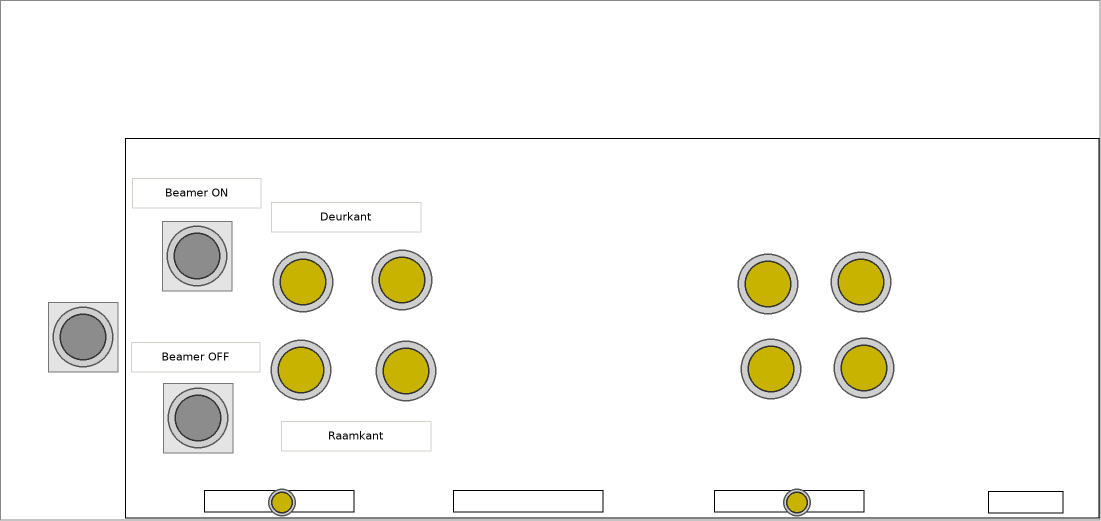
VISUALIZATION Visualization  // 1101x521
    Rectangle (125,138 974x380)
    Lamp1 (268,247 70x70), variable: Lichtsturing.relaisstandDEUR, style: Lamp-Lamp1-Yellow
    Lamp1 (367,245 70x70), variable: Lichtsturing.relaisstandDEUR, style: Lamp-Lamp1-Yellow
    Lamp1 (733,249 70x70), variable: Lichtsturing.relaisstandDEUR, style: Lamp-Lamp1-Yellow
    Lamp1 (826,247 70x70), variable: Lichtsturing.relaisstandDEUR, style: Lamp-Lamp1-Yellow
    Lamp1 (266,335 70x70), variable: Lichtsturing.relaisstandRAAM, style: Lamp-Lamp1-Yellow
    Lamp1 (371,336 70x70), variable: Lichtsturing.relaisstandRAAM, style: Lamp-Lamp1-Yellow
    Lamp1 (736,334 70x70), variable: Lichtsturing.relaisstandRAAM, style: Lamp-Lamp1-Yellow
    Lamp1 (829,333 70x70), variable: Lichtsturing.relaisstandRAAM, style: Lamp-Lamp1-Yellow
    Rectangle (204,490 150x22)
    Rectangle (453,490 150x22)
    Rectangle (714,490 150x22)
    Rectangle (988,491 75x22)
    Lamp1 (266,486 32x33), variable: EnOcean.raam2open, style: Lamp-Lamp1-Yellow
    Lamp1 (781,486 32x33), variable: EnOcean.raam1open, style: Lamp-Lamp1-Yellow
    Textfield (271,202 150x30), "Deurkant"
    Textfield (281,421 150x30), "Raamkant"
    PushSwitch (162,221 70x70), variable: BeamerAANKNOP, behaviour: TOGGLE, style: Switch-PushSwitch-Gray
    Textfield (132,178 129x30), "Beamer ON"
    PushSwitch (163,383 70x70), variable: BeamerUITKNOP, behaviour: TOGGLE, style: Switch-PushSwitch-Gray
    Textfield (131,342 129x30), "Beamer OFF"
    PushSwitch (48,302 70x70), variable: Beamercontrol.bconnect, behaviour: TOGGLE, style: Switch-PushSwitch-Gray
END_VISUALIZATION

(* stored: Version 1.1.0.1, ProductVersion 3.1.4022.10
   Visu Visualization: Id {8a15400c-277f-4c6e-aa9a-e38930a493bf} *)
